ABB RobotStudio station: ROS_20171103-125232.rsstn

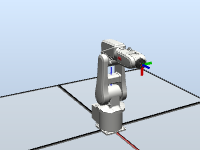
Station ROS (saved by RobotStudio 6.6.7603.115)
Controller ABB_IRB_120_ROS
  mechanical unit ROB_1: IRB120_3_58__01, 6 joints, base frame (0, 0, 0) mm
Layout (positions relative to the parent item):
  - IRB120_3_58__01 [mechanism, from Robots\IRB120_3_58_G_01.rslib] at (0, 0, 0) mm; joint values [0, 0, 0, 0, 0, 0] (rad or m)
